TYPE ST_UPSEvents :
STRUCT
	b_BatteryLowNotice		:	BOOL;	//initialize DC conditioning
	b_BatteryLowWarning		:	BOOL;	//Battery charging failed, consider shutdown
	b_BatteryLowError		:	BOOL;	//Battery level critical, System should shutdown
	b_NoBatteryError		:	BOOL;	//no Battery voltage detected?
	b_InputVoltageError		:	BOOL;	//ipsstate says 24v is available, but no input is seen.
END_STRUCT
END_TYPE

(* stored: Version 1.1.0.1, ProductVersion 3.1.4024.12
   DUT ST_UPSEvents: Id {2075b0c0-1330-4f6b-9861-c97a9d769a04} *)
